{attribute 'qualified_only'}
TYPE E_SDSGarageRStates :
(
    UNKNOWN := 0,
    T1 := 1,
    T2 := 2,
    T3 := 3,
    T4 := 4,
    M1 := 5,
    M2 := 6,
    M3 := 7,
    M4 := 8,
    B1 := 9,
    B2 := 10,
    B3 := 11,
    B4 := 12,
    PREDICTED_HOME := 13
) UINT;
END_TYPE

(* stored: Version 1.1.0.1
   DUT E_SDSGarageRStates: Id {f0733f68-1a1b-0d48-055a-00195f147a77} *)
